FUNCTION_BLOCK LowTemperatureHeatingNetwork
VAR_INPUT
END_VAR
VAR_OUTPUT
END_VAR
VAR
END_VAR

END_FUNCTION_BLOCK

(* stored: Version 1.1.0.1, ProductVersion 3.1.4024.10
   POU LowTemperatureHeatingNetwork: Id {41e3edb3-66e7-411c-a35e-b44e9a5d66f1}, SpecialFunc None *)
